PROGRAM MAIN
VAR
	(* JSON *)
	fbJson 			: FB_JsonDomParser;
	jsonDoc 		: SJsonValue;
	jsonProp		: SJsonValue;
	jsonValue		: SJsonValue;
	bHasMember		: BOOL;
  	sMessage 		: STRING(255) := '{"serialNumber":"G030PT028191AC4R","batteryVoltage":"1547mV","clickType":"SINGLE"}';
	stReceivedData	: ST_ReceivedData;
END_VAR

(* Retrieve JSON content *)
jsonDoc := fbJson.ParseDocument(sMessage);
bHasMember := fbJson.HasMember(jsonDoc, 'serialNumber');
IF (bHasMember) THEN
	  bHasMember := FALSE;
	  jsonProp := fbJson.FindMember(jsonDoc, 'serialNumber');
	  stReceivedData.serialNumber := fbJson.GetString(jsonProp);
END_IF

bHasMember := fbJson.HasMember(jsonDoc, 'batteryVoltage');
IF (bHasMember) THEN
	  bHasMember := FALSE;
	  jsonProp := fbJson.FindMember(jsonDoc, 'batteryVoltage');
	  stReceivedData.batteryVoltage := fbJson.GetString(jsonProp);
END_IF		

bHasMember := fbJson.HasMember(jsonDoc, 'clickType');
IF (bHasMember) THEN
	  bHasMember := FALSE;
	  jsonProp := fbJson.FindMember(jsonDoc, 'clickType');
	  stReceivedData.clickType := fbJson.GetString(jsonProp);
END_IF

END_PROGRAM

(* stored: Version 1.1.0.1, ProductVersion 3.1.4022.3
   POU MAIN: Id {d584e34a-6630-44df-b26c-54c4ec0ec00a}, SpecialFunc None *)
